PROGRAM MAIN
VAR
	tcpTest : FB_TcpSendReceivingQueue;
	tcpTest2 : FB_TcpSendReceiving;
	bAddTask: BOOL;
	arrData : ARRAY[0..255] OF BYTE;
	arrRecv : ARRAY[0..255] OF BYTE;
	bool1 : BOOL;
	bool2 : BOOL;
	dint1 : DINT;
	dint2 :DINT;
	STR1:STRING;
	MD5 : ARRAY[0..31] OF BYTE;
	MD5STR : STRING;
END_VAR

F_GenerateHashValue(
	hashMode:= Tc2_Utilities.E_HashMode.HASH_MD5, 
	pData:= ADR(STR1), 
	nData:= LEN(STR1), 
	pHash:= ADR(MD5), 
	nHash:= 16);
// 测试同时向两个仓库推送2
dint1 := 2030/100;
dint2 := 2030 MOD 100;
bool1 := FAILED(0);
bool2 := FAILED(16#80000013);
IF bAddTask THEN
	bAddTask := FALSE;
	arrData[0] := 67;
	tcpTest.AddTask('Send', 0, ADR(arrData), SIZEOF(arrData));
	tcpTest.AddTask('Send', 0, ADR(arrData), SIZEOF(arrData));
	tcpTest.AddTask('Send', 0, ADR(arrData), SIZEOF(arrData));
	tcpTest.AddTask('Send', 0, ADR(arrData), SIZEOF(arrData));
	tcpTest.AddTask('Send', 0, ADR(arrData), SIZEOF(arrData));
	arrData[0] := 68;
	tcpTest.AddTask('Send', 0, ADR(arrData), SIZEOF(arrData));
	tcpTest.AddTask('Send', 0, ADR(arrData), SIZEOF(arrData));
	tcpTest.AddTask('Send', 0, ADR(arrData), SIZEOF(arrData));
	tcpTest.AddTask('Send', 0, ADR(arrData), SIZEOF(arrData));
	tcpTest.AddTask('Send', 0, ADR(arrData), SIZEOF(arrData));
	arrData[0] := 69;
	tcpTest.AddTask('Send', 0, ADR(arrData), SIZEOF(arrData));
	tcpTest.AddTask('Send', 0, ADR(arrData), SIZEOF(arrData));
	tcpTest.AddTask('Send', 0, ADR(arrData), SIZEOF(arrData));
	tcpTest.AddTask('Send', 0, ADR(arrData), SIZEOF(arrData));
	tcpTest.AddTask('Send', 0, ADR(arrData), SIZEOF(arrData));
	arrData[0] := 70;
	tcpTest.AddTask('Send', 0, ADR(arrData), SIZEOF(arrData));
	tcpTest.AddTask('Send', 0, ADR(arrData), SIZEOF(arrData));
	tcpTest.AddTask('Send', 0, ADR(arrData), SIZEOF(arrData));
	tcpTest.AddTask('Send', 0, ADR(arrData), SIZEOF(arrData));
	tcpTest.AddTask('Send', 0, ADR(arrData), SIZEOF(arrData));
	arrData[0] := 71;
	tcpTest.AddTask('Send', 0, ADR(arrData), SIZEOF(arrData));
	tcpTest.AddTask('Send', 0, ADR(arrData), SIZEOF(arrData));
	tcpTest.AddTask('Send', 0, ADR(arrData), SIZEOF(arrData));
	tcpTest.AddTask('Send', 0, ADR(arrData), SIZEOF(arrData));
	tcpTest.AddTask('Send', 0, ADR(arrData), SIZEOF(arrData));
	arrData[0] := 72;
	tcpTest.AddTask('Send', 0, ADR(arrData), SIZEOF(arrData));
	tcpTest.AddTask('Send', 0, ADR(arrData), SIZEOF(arrData));
	tcpTest.AddTask('Send', 0, ADR(arrData), SIZEOF(arrData));
	tcpTest.AddTask('Send', 0, ADR(arrData), SIZEOF(arrData));
	tcpTest.AddTask('Send', 0, ADR(arrData), SIZEOF(arrData));
	arrData[0] := 73;
	tcpTest.AddTask('Send', 0, ADR(arrData), SIZEOF(arrData));
	tcpTest.AddTask('Send', 0, ADR(arrData), SIZEOF(arrData));
	tcpTest.AddTask('Send', 0, ADR(arrData), SIZEOF(arrData));
	tcpTest.AddTask('Send', 0, ADR(arrData), SIZEOF(arrData));
	tcpTest.AddTask('Send', 0, ADR(arrData), SIZEOF(arrData));
	arrData[0] := 74;
	tcpTest.AddTask('Send', 0, ADR(arrData), SIZEOF(arrData));
	tcpTest.AddTask('Send', 0, ADR(arrData), SIZEOF(arrData));
	tcpTest.AddTask('Send', 0, ADR(arrData), SIZEOF(arrData));
	tcpTest.AddTask('Send', 0, ADR(arrData), SIZEOF(arrData));
	tcpTest.AddTask('Send', 0, ADR(arrData), SIZEOF(arrData));
END_IF
tcpTest(
	bEnable:= TRUE, 
	bReset:= , 
	sRemoteIp:= '127.0.0.1', 
	nRemotePort:= 8003, 
	pRecvData:= ADR(arrRecv), 
	nRecvSize:= SIZEOF(arrRecv), 
	bBusyConnect=> , 
	bConnected=> , 
	bBusySend=> , 
	bSendDone=> , 
	bBusyRecv=> , 
	bRecvDone=> , 
	bError=> , 
	nRecvBytes=> , 
	bDataReceived=> );

END_PROGRAM

(* stored: Version 1.1.0.1, ProductVersion 3.1.4024.12
   POU MAIN: Id {5acbb519-50b6-4a11-9b3f-9b411aa3ed7d}, SpecialFunc None *)
